// TIA Portal V20 export
TYPE "TypeWenglorP3PC301Sd"
   STRUCT
      LaserOff : Bool;   // Laser off (1=Off)
      Localization : Bool;   // Localization (1=On)
      res2 : Bool;
      SCC1TeachIn : Bool;   // Start Teach SCC1
      SCC2TeachIn : Bool;   // Start Teach SCC2
      res5 : Bool;
      res6 : Bool;
      res7 : Bool;
   END_STRUCT;
END_TYPE
